// TIA Portal V18 export
DATA_BLOCK "IO_Settings"   // DB101
{ S7_Optimized_Access := 'TRUE' }
// This datablock will hold the IO setup settings for the unit
// stored: AutoNumber false, MemoryReserve 100
   VAR RETAIN
      ChargePress1Tx { S7_SetPoint := 'True'} : Bool;   // Charge Pressure Transducer Exist - used for alarms
      ChargePress1Sw { S7_SetPoint := 'True'} : Bool;
      ChargePress2Tx { S7_SetPoint := 'True'} : Bool;   // Charge Pressure Transducer Exist - used for alarms
      ChargePress2Sw { S7_SetPoint := 'True'} : Bool;
      SecondaryFilters { S7_SetPoint := 'True'} : Bool;   // Set bit if 2 FWD and REV filters exist.
      HPUType { S7_SetPoint := 'True'} : Int;   // 0 = Elec HPU , 1 = CAT HPU
      LubeFlowSwitch { S7_SetPoint := 'True'} : Bool;   // Set if TD is equiped with Lube Flow Switch
      KLoopFilter { S7_SetPoint := 'True'} : Bool;   // Set if KL Filter is equipped
      ElevClSw { S7_SetPoint := 'True'} : Bool;   // Set if Elevator Close Switch exists
   END_VAR
BEGIN
END_DATA_BLOCK
